    fTable_Si : ARRAY[0..755, 0..2] OF LREAL := [
        10.0000, -9999, 3.94851,
        10.1617, -9999, 3.95531,
        10.3261, -9999, 3.96212,
        10.4931, -9999, 3.96894,
        10.6628, -9999, 3.97577,
        10.8353, -9999, 3.98262,
        11.0105, -9999, 3.98948,
        11.1886, -9999, 3.99635,
        11.3696, -9999, 4.00322,
        11.5535, -9999, 4.01012,
        11.7404, -9999, 4.01702,
        11.9303, -9999, 4.02394,
        12.1232, -9999, 4.00019,
        12.3193, -9999, 3.95930,
        12.5186, -9999, 3.91883,
        12.7210, -9999, 3.87876,
        12.9268, -9999, 3.83911,
        13.1359, -9999, 3.79987,
        13.3483, -9999, 3.76102,
        13.5642, -9999, 3.72257,
        13.7836, -9999, 3.68452,
        14.0066, -9999, 3.64513,
        14.2331, -9999, 3.55020,
        14.4633, -9999, 3.45774,
        14.6972, -9999, 3.36769,
        14.9350, -9999, 3.27998,
        15.1765, -9999, 3.19455,
        15.4220, -9999, 3.11136,
        15.6714, -9999, 3.03032,
        15.9249, -9999, 2.95140,
        16.1825, -9999, 2.83114,
        16.4442, -9999, 2.69869,
        16.7102, -9999, 2.57244,
        16.9805, -9999, 2.45210,
        17.2551, -9999, 2.33738,
        17.5342, -9999, 2.22803,
        17.8178, -9999, 2.12380,
        18.1060, -9999, 1.97554,
        18.3988, -9999, 1.76138,
        18.6964, -9999, 1.57043,
        18.9988, -9999, 1.40019,
        19.3061, -9999, 1.24840,
        19.6184, -9999, 1.11306,
        19.9357, -9999, 0.992396,
        20.2581, -9999, 0.862336,
        20.5858, -9999, 0.753564,
        20.9187, -9999, 0.698871,
        21.2571, -9999, 0.648148,
        21.6009, -9999, 0.602543,
        21.9503, -9999, 0.561516,
        22.3053, -9999, 0.523281,
        22.6661, -9999, 0.496895,
        23.0327, -9999, 0.478071,
        23.4052, -9999, 0.459962,
        23.7838, -9999, 0.442538,
        24.1685, -9999, 0.425774,
        24.5594, -9999, 0.413096,
        24.9566, -9999, 0.403041,
        25.3602, -9999, 0.393231,
        25.7704, -9999, 0.383660,
        26.1872, -9999, 0.374321,
        26.6108, -9999, 0.365210,
        27.0412, -9999, 0.366288,
        27.4786, -9999, 0.367374,
        27.9230, -9999, 0.368463,
        28.3747, -9999, 0.369555,
        28.8336, -9999, 0.370650,
        29.3000, 3.83380, 0.371749,
        29.7739, 3.80691, 0.372851,
        30.2554, 3.78097, 0.373956,
        30.7448, 3.75582, 0.375064,
        31.2421, 3.73048, 0.376176,
        31.7474, 3.70550, 0.378088,
        32.2609, 3.68147, 0.381996,
        32.7827, 3.65905, 0.385945,
        33.3129, 3.63764, 0.389935,
        33.8517, 3.61703, 0.393965,
        34.3992, 3.59711, 0.398038,
        34.9556, 3.57779, 0.402152,
        35.5210, 3.55900, 0.406309,
        36.0955, 3.54071, 0.410509,
        36.6793, 3.52286, 0.414753,
        37.2726, 3.50545, 0.419040,
        37.8754, 3.48848, 0.423372,
        38.4880, 3.47200, 0.427748,
        39.1106, 3.45628, 0.432170,
        39.7431, 3.44176, 0.435537,
        40.3860, 3.42689, 0.437136,
        41.0392, 3.41050, 0.438741,
        41.7029, 3.39378, 0.440351,
        42.3774, 3.37667, 0.441968,
        43.0629, 3.35917, 0.443590,
        43.7594, 3.34130, 0.445218,
        44.4671, 3.32304, 0.446852,
        45.1864, 3.30440, 0.448493,
        45.9172, 3.28549, 0.450139,
        46.6599, 3.26615, 0.451198,
        47.4146, 3.24599, 0.451979,
        48.1815, 3.22476, 0.452762,
        48.9608, 3.20267, 0.453547,
        49.7527, 3.17964, 0.454332,
        50.5574, 3.15558, 0.455119,
        51.3751, 3.13042, 0.455908,
        52.2061, 3.10325, 0.456698,
        53.0505, 3.07444, 0.458301,
        53.9085, 3.04507, 0.461948,
        54.7804, 3.01545, 0.465624,
        55.6665, 2.98498, 0.469328,
        56.5668, 2.95338, 0.473062,
        57.4817, 2.92040, 0.476826,
        58.4115, 2.88519, 0.480620,
        59.3562, 2.84598, 0.484444,
        60.3163, 2.80606, 0.494947,
        61.2918, 2.76788, 0.506504,
        62.2832, 2.73042, 0.518332,
        63.2906, 2.69333, 0.530436,
        64.3142, 2.65696, 0.542822,
        65.3545, 2.62418, 0.554884,
        66.4115, 2.58874, 0.558968,
        67.4857, 2.54971, 0.563081,
        68.5772, 2.50917, 0.567224,
        69.6864, 2.46935, 0.571398,
        70.8135, 2.43129, 0.566814,
        71.9588, 2.38275, 0.552979,
        73.1227, 2.32504, 0.539483,
        74.3054, 2.26322, 0.526316,
        75.5072, 2.19828, 0.504782,
        76.7285, 2.11635, 0.477417,
        77.9695, 2.01618, 0.451535,
        79.2306, 1.90170, 0.427364,
        80.5121, 1.77437, 0.422623,
        81.8143, 1.64458, 0.417936,
        83.1376, 1.50518, 0.413300,
        84.4823, 1.34727, 0.409326,
        85.8487, 1.17621, 0.415946,
        87.2373, 0.995339, 0.422674,
        88.6483, 0.794497, 0.429510,
        90.0821, 0.568059, 0.436457,
        91.5391, 0.306962, 0.444926,
        93.0197, 0.00161588, 0.456528,
        94.5242, -0.366911, 0.468434,
        96.0530, -0.841388, 0.480650,
        97.6066, -1.52605, 0.495035,
        99.1853, -2.88115, 0.517644,
        99.5000, -3.50392, 0.522228,
        99.5240, -3.56793, 0.517644,
        99.5490, -3.65086, 0.517841,
        99.5760, -3.74861, 0.521284,
        99.6010, -3.84977, 0.535297,
        99.6260, -3.95788, 0.552022,
        99.6490, -4.07048, 0.581748,
        99.6760, -4.21370, 0.630001,
        99.6990, -4.33738, 0.708784,
        99.7260, -4.47439, 0.813415,
        99.7490, -4.57087, 0.941569,
        99.7750, -4.65499, 1.07721,
        99.8260, -4.76959, 1.37513,
        99.8510, -4.79109, 1.52203,
        99.8750, -4.78699, 1.65993,
        99.8990, -4.76674, 1.77995,
        99.9260, -4.73984, 1.87968,
        99.9510, -4.72571, 1.97448,
        99.9740, -4.69897, 2.05815,
        100.000, -4.67405, 2.13311,
        100.030, -4.65490, 2.20171,
        100.120, -4.60024, 2.41667,
        100.180, -4.60059, 2.49729,
        100.220, -4.62085, 2.58505,
        100.250, -4.64510, 2.62089,
        100.280, -4.70275, 2.67241,
        100.300, -4.73916, 2.73072,
        100.350, -4.82406, 2.91360,
        100.380, -4.87754, 3.01959,
        100.450, -4.89461, 3.39622,
        100.480, -4.89177, 3.52655,
        100.500, -4.87133, 3.64732,
        100.550, -4.80557, 3.86847,
        100.600, -4.71048, 4.10668,
        100.620, -4.63514, 4.23678,
        100.680, -4.54337, 4.36464,
        100.700, -4.48607, 4.49509,
        100.750, -4.33702, 4.75764,
        100.770, -4.23325, 4.85961,
        100.800, -4.07337, 4.94637,
        100.850, -3.81798, 5.07430,
        100.900, -3.56548, 5.12335,
        101.000, -3.15785, 5.13032,
        101.020, -3.08861, 5.12048,
        101.250, -2.52100, 5.15904,
        101.320, -2.30405, 5.19959,
        101.380, -2.08534, 5.20146,
        101.400, -2.00971, 5.18989,
        101.450, -1.81270, 5.13442,
        101.500, -1.65152, 5.02977,
        101.600, -1.41105, 4.78618,
        101.630, -1.36359, 4.72648,
        101.650, -1.35292, 4.65861,
        101.750, -1.25455, 4.44125,
        101.820, -1.21389, 4.30165,
        101.880, -1.19458, 4.18620,
        101.900, -1.20985, 4.13288,
        101.950, -1.20581, 4.08850,
        102.000, -1.19801, 3.97606,
        102.030, -1.22710, 3.93010,
        102.050, -1.24904, 3.89784,
        102.100, -1.28103, 3.86731,
        102.150, -1.30990, 3.80579,
        102.180, -1.33991, 3.78427,
        102.250, -1.39700, 3.76802,
        102.300, -1.42608, 3.74849,
        102.350, -1.46728, 3.74261,
        102.400, -1.50309, 3.76084,
        102.450, -1.52538, 3.79386,
        102.530, -1.50608, 3.87484,
        102.550, -1.48153, 3.89373,
        102.600, -1.42009, 3.90179,
        102.650, -1.36279, 3.88239,
        102.700, -1.31820, 3.83958,
        102.780, -1.29202, 3.76416,
        102.880, -1.29963, 3.67993,
        102.950, -1.32951, 3.64539,
        103.000, -1.34633, 3.63286,
        103.120, -1.36198, 3.65919,
        103.200, -1.32264, 3.65521,
        103.280, -1.27117, 3.62578,
        103.320, -1.25882, 3.57767,
        103.350, -1.24200, 3.56029,
        103.430, -1.23327, 3.47903,
        103.450, -1.26147, 3.44200,
        103.550, -1.32267, 3.37538,
        103.600, -1.36022, 3.35329,
        103.620, -1.37658, 3.35242,
        103.700, -1.42690, 3.33036,
        103.800, -1.48061, 3.33205,
        103.880, -1.50969, 3.33940,
        104.000, -1.53630, 3.33472,
        104.100, -1.56167, 3.31576,
        104.220, -1.62193, 3.27368,
        104.280, -1.65400, 3.27417,
        104.430, -1.72694, 3.28606,
        104.470, -1.75387, 3.27978,
        104.500, -1.76829, 3.28791,
        104.530, -1.78693, 3.28885,
        104.570, -1.80294, 3.29751,
        104.650, -1.83679, 3.30856,
        104.730, -1.87270, 3.30556,
        104.750, -1.88124, 3.31109,
        104.800, -1.90801, 3.30176,
        104.900, -1.98706, 3.33116,
        104.930, -2.00067, 3.33359,
        104.950, -2.00298, 3.34991,
        105.030, -2.04570, 3.36298,
        105.150, -2.11934, 3.39504,
        105.180, -2.13949, 3.40977,
        105.250, -2.17952, 3.43515,
        105.320, -2.21343, 3.47153,
        105.350, -2.23848, 3.47688,
        105.430, -2.28483, 3.52378,
        105.500, -2.32999, 3.56457,
        105.550, -2.35832, 3.60198,
        105.600, -2.38578, 3.64781,
        105.630, -2.39089, 3.66569,
        105.750, -2.44861, 3.77644,
        105.780, -2.45326, 3.79743,
        105.850, -2.48245, 3.88408,
        105.870, -2.48052, 3.91584,
        105.970, -2.42689, 4.01616,
        106.030, -2.39972, 4.04717,
        106.070, -2.38240, 4.06604,
        106.100, -2.37398, 4.06874,
        106.230, -2.38361, 4.11947,
        106.270, -2.37996, 4.15308,
        106.320, -2.37462, 4.16809,
        106.400, -2.36004, 4.21391,
        106.430, -2.36196, 4.22064,
        106.450, -2.36509, 4.23983,
        106.550, -2.33925, 4.28215,
        106.620, -2.33379, 4.30894,
        106.650, -2.33507, 4.32546,
        106.700, -2.32865, 4.34622,
        106.750, -2.32543, 4.37918,
        106.800, -2.31100, 4.39528,
        106.870, -2.30275, 4.43789,
        106.920, -2.28031, 4.45074,
        106.970, -2.27262, 4.47446,
        107.000, -2.25035, 4.47193,
        107.150, -2.24976, 4.52075,
        107.170, -2.23267, 4.52195,
        107.200, -2.22431, 4.53560,
        107.280, -2.22372, 4.53468,
        107.300, -2.22218, 4.54692,
        107.320, -2.21789, 4.54827,
        107.350, -2.21747, 4.55993,
        107.400, -2.22568, 4.56521,
        107.420, -2.21201, 4.58499,
        107.500, -2.21196, 4.60002,
        107.530, -2.21439, 4.60834,
        107.550, -2.21478, 4.62406,
        107.580, -2.20227, 4.63210,
        107.600, -2.20862, 4.62922,
        107.620, -2.19987, 4.64804,
        107.670, -2.19745, 4.66695,
        107.730, -2.18227, 4.67472,
        107.750, -2.19300, 4.68717,
        107.850, -2.17068, 4.70239,
        107.880, -2.18424, 4.71832,
        107.930, -2.18294, 4.73505,
        107.950, -2.19199, 4.75539,
        108.070, -2.15772, 4.79660,
        108.220, -2.13084, 4.82955,
        108.280, -2.11240, 4.85593,
        108.420, -2.08897, 4.88059,
        108.450, -2.08958, 4.88346,
        108.520, -2.07611, 4.91320,
        108.570, -2.06068, 4.91793,
        108.600, -2.05985, 4.93016,
        108.730, -2.02793, 4.92866,
        108.830, -2.03087, 4.94162,
        108.900, -2.01993, 4.96783,
        109.000, -1.99875, 4.97239,
        109.030, -1.99361, 4.97267,
        109.070, -1.99579, 4.95935,
        109.120, -2.00066, 4.97576,
        109.200, -2.00421, 4.98276,
        109.250, -1.99981, 4.99897,
        109.270, -1.98698, 4.98829,
        109.350, -2.00603, 4.99135,
        109.380, -2.00850, 4.98316,
        109.400, -2.01211, 4.99342,
        109.430, -2.02183, 4.98967,
        109.450, -2.01515, 5.00593,
        109.530, -2.04292, 5.01580,
        109.550, -2.03376, 5.03141,
        109.570, -2.03838, 5.02656,
        109.600, -2.03677, 5.04483,
        109.620, -2.03705, 5.03873,
        109.670, -2.02773, 5.05325,
        109.800, -2.05572, 5.08673,
        109.970, -2.05841, 5.12220,
        110.000, -2.08477, 5.13791,
        110.500, -2.08318, 5.28267,
        111.000, -2.07105, 5.45779,
        111.500, -2.02987, 5.61544,
        112.500, -1.94845, 5.85909,
        114.000, -1.92517, 6.16450,
        114.500, -1.96395, 6.33338,
        115.000, -1.98987, 6.51862,
        115.500, -1.96320, 6.72312,
        117.000, -1.77809, 7.40254,
        117.500, -1.61173, 7.59488,
        118.000, -1.45934, 7.77180,
        118.500, -1.28616, 7.87553,
        119.000, -1.13984, 8.02234,
        119.500, -0.959918, 8.05843,
        121.433, -0.578394, 8.42371,
        121.500, -0.573231, 8.43660,
        122.000, -0.405651, 8.51447,
        123.500, -0.0264126, 8.67192,
        124.000, 0.0779155, 8.69958,
        124.500, 0.171345, 8.77704,
        125.000, 0.293945, 8.78726,
        127.000, 0.572464, 9.00076,
        127.500, 0.671836, 9.04215,
        128.500, 0.827038, 9.19455,
        129.500, 0.995074, 9.33439,
        130.000, 1.11832, 9.43724,
        131.500, 1.53131, 9.68832,
        133.000, 2.07611, 9.80683,
        133.500, 2.28741, 9.78221,
        134.500, 2.61972, 9.60861,
        136.000, 2.84736, 9.24827,
        136.500, 2.87943, 9.17385,
        137.000, 2.87745, 9.11857,
        137.500, 2.85152, 9.03612,
        139.500, 2.83348, 9.09883,
        140.000, 2.84307, 9.12631,
        140.500, 2.88384, 9.18357,
        141.500, 3.00310, 9.19764,
        142.000, 3.03093, 9.17508,
        142.500, 3.03358, 9.18522,
        143.000, 3.03374, 9.17393,
        144.000, 3.03215, 9.32209,
        145.000, 3.09900, 9.41818,
        145.500, 3.16288, 9.49844,
        146.000, 3.22259, 9.51997,
        146.500, 3.28049, 9.57995,
        147.000, 3.34172, 9.60862,
        147.500, 3.41479, 9.66258,
        148.000, 3.48151, 9.67350,
        148.500, 3.56199, 9.71113,
        149.500, 3.68256, 9.71835,
        150.000, 3.70254, 9.69979,
        150.500, 3.68373, 9.74096,
        151.000, 3.69207, 9.84710,
        151.500, 3.76904, 10.0037,
        152.000, 3.94900, 10.1180,
        152.500, 4.15147, 10.1431,
        153.500, 4.47402, 9.96424,
        154.500, 4.52214, 9.69132,
        155.000, 4.47788, 9.64167,
        155.500, 4.41664, 9.63644,
        156.000, 4.38177, 9.66128,
        156.500, 4.35929, 9.73288,
        157.500, 4.39020, 9.79855,
        158.000, 4.36737, 9.87036,
        158.500, 4.42951, 9.99628,
        159.000, 4.48663, 9.99841,
        160.000, 4.57954, 10.1071,
        162.500, 4.84589, 10.5019,
        163.500, 5.05409, 10.6336,
        164.500, 5.27583, 10.7324,
        165.500, 5.50795, 10.7656,
        166.500, 5.73389, 10.8239,
        167.000, 5.79695, 10.7800,
        167.500, 5.86489, 10.9015,
        169.000, 6.35522, 10.9520,
        170.000, 6.66644, 10.9210,
        171.500, 7.13398, 10.7554,
        172.000, 7.24279, 10.5495,
        172.500, 7.29281, 10.5369,
        173.000, 7.38343, 10.4391,
        173.500, 7.52303, 10.4208,
        174.000, 7.60600, 10.1923,
        174.500, 7.64212, 10.1249,
        175.000, 7.66842, 9.98038,
        176.000, 7.68591, 9.82584,
        176.500, 7.67332, 9.72546,
        177.000, 7.68563, 9.66145,
        178.000, 7.67511, 9.60542,
        178.500, 7.69740, 9.51565,
        179.000, 7.64095, 9.49283,
        179.500, 7.63925, 9.43704,
        179.990, 7.55398, 9.49765,
        182.901, 7.85149, 9.42072,
        185.859, 7.94847, 9.34442,
        188.866, 8.10574, 9.26640,
        191.920, 8.27005, 9.17918,
        195.025, 8.43202, 9.09278,
        198.179, 8.59128, 9.00719,
        201.384, 8.74251, 8.92241,
        204.641, 8.88646, 8.85010,
        207.951, 9.03960, 8.78533,
        211.315, 9.19861, 8.72104,
        214.733, 9.36085, 8.65722,
        218.206, 9.53668, 8.59386,
        221.735, 9.72509, 8.52313,
        225.322, 9.90451, 8.41115,
        228.966, 10.0644, 8.30065,
        232.669, 10.2142, 8.19159,
        236.432, 10.3574, 8.08397,
        240.257, 10.4958, 7.97776,
        244.143, 10.6314, 7.87295,
        248.091, 10.7716, 7.76952,
        252.104, 10.9063, 7.65024,
        256.182, 11.0283, 7.53005,
        260.325, 11.1426, 7.41174,
        264.536, 11.2509, 7.29529,
        268.814, 11.3543, 7.18067,
        273.162, 11.4535, 7.06784,
        277.580, 11.5489, 6.95680,
        282.070, 11.6411, 6.84750,
        286.632, 11.7306, 6.73991,
        291.268, 11.8181, 6.63402,
        295.979, 11.9057, 6.52979,
        300.767, 11.9918, 6.42157,
        305.631, 12.0733, 6.31071,
        310.575, 12.1486, 6.20175,
        315.598, 12.2203, 6.09469,
        320.702, 12.2889, 5.98947,
        325.890, 12.3551, 5.88607,
        331.161, 12.4191, 5.78445,
        336.517, 12.4812, 5.68459,
        341.960, 12.5420, 5.58645,
        347.491, 12.6018, 5.49000,
        353.111, 12.6614, 5.39523,
        358.822, 12.7222, 5.30208,
        364.626, 12.7889, 5.21055,
        370.523, 12.8576, 5.10056,
        376.516, 12.9142, 4.98768,
        382.606, 12.9608, 4.87731,
        388.795, 13.0027, 4.76937,
        395.083, 13.0407, 4.66382,
        401.473, 13.0753, 4.56061,
        407.967, 13.1069, 4.45967,
        414.565, 13.1360, 4.36098,
        421.270, 13.1628, 4.26447,
        428.084, 13.1876, 4.17009,
        435.008, 13.2107, 4.07781,
        442.044, 13.2322, 3.98756,
        449.194, 13.2527, 3.89931,
        456.459, 13.2727, 3.81302,
        463.842, 13.2933, 3.72727,
        471.344, 13.3117, 3.63809,
        478.968, 13.3260, 3.55105,
        486.715, 13.3375, 3.46608,
        494.587, 13.3472, 3.38316,
        502.587, 13.3552, 3.30221,
        510.715, 13.3617, 3.22320,
        518.976, 13.3670, 3.14609,
        527.370, 13.3711, 3.07081,
        535.900, 13.3742, 2.99734,
        544.567, 13.3764, 2.92563,
        553.375, 13.3779, 2.85563,
        562.326, 13.3789, 2.78730,
        571.421, 13.3797, 2.72061,
        580.663, 13.3815, 2.65552,
        590.055, 13.3832, 2.58813,
        599.599, 13.3823, 2.52006,
        609.297, 13.3786, 2.45378,
        619.151, 13.3731, 2.38925,
        629.166, 13.3663, 2.32641,
        639.342, 13.3582, 2.26522,
        649.683, 13.3491, 2.20565,
        660.191, 13.3390, 2.14764,
        670.869, 13.3278, 2.09115,
        681.720, 13.3158, 2.03616,
        692.746, 13.3006, 1.98261,
        703.951, 13.2845, 1.93392,
        715.336, 13.2706, 1.88812,
        726.906, 13.2578, 1.84339,
        738.664, 13.2453, 1.79973,
        750.611, 13.2332, 1.75710,
        762.751, 13.2215, 1.71548,
        775.088, 13.2102, 1.67484,
        787.625, 13.1996, 1.63517,
        800.364, 13.1912, 1.59508,
        813.309, 13.1807, 1.55256,
        826.464, 13.1685, 1.51118,
        839.831, 13.1555, 1.47089,
        853.415, 13.1418, 1.43168,
        867.218, 13.1278, 1.39352,
        881.245, 13.1136, 1.35637,
        895.498, 13.1001, 1.32021,
        909.982, 13.0874, 1.28196,
        924.700, 13.0717, 1.24308,
        939.656, 13.0542, 1.20538,
        954.855, 13.0353, 1.16882,
        970.299, 13.0154, 1.13337,
        985.992, 12.9946, 1.09899,
        1001.94, 12.9729, 1.06561,
        1018.15, 12.9502, 1.03318,
        1034.61, 12.9266, 1.00174,
        1051.35, 12.9020, 0.971249,
        1068.35, 12.8761, 0.941688,
        1085.63, 12.8487, 0.913028,
        1103.19, 12.8192, 0.887547,
        1121.03, 12.7911, 0.864407,
        1139.17, 12.7632, 0.841817,
        1157.59, 12.7350, 0.819826,
        1176.31, 12.7063, 0.798411,
        1195.34, 12.6771, 0.777531,
        1214.67, 12.6470, 0.757139,
        1234.32, 12.6159, 0.737234,
        1254.28, 12.5837, 0.717856,
        1274.57, 12.5503, 0.698989,
        1295.19, 12.5156, 0.680609,
        1316.13, 12.4792, 0.662552,
        1337.42, 12.4409, 0.644954,
        1359.05, 12.4006, 0.627806,
        1381.04, 12.3579, 0.611117,
        1403.37, 12.3125, 0.594814,
        1426.07, 12.2640, 0.578892,
        1449.14, 12.2120, 0.563357,
        1472.58, 12.1559, 0.548240,
        1496.39, 12.0950, 0.533519,
        1520.60, 12.0284, 0.518512,
        1545.19, 11.9546, 0.503884,
        1570.18, 11.8721, 0.489627,
        1595.58, 11.7790, 0.475781,
        1621.39, 11.6727, 0.462322,
        1647.61, 11.5493, 0.449240,
        1674.26, 11.4029, 0.436529,
        1701.34, 11.2243, 0.424180,
        1728.86, 10.9982, 0.412181,
        1756.82, 10.6935, 0.399995,
        1785.24, 10.2377, 0.388066,
        1814.11, 9.37942, 0.376400,
        1815, 9.33435, 0.376049,
        1838.80, 2.82013, 0.366843,
        1839, 2.82204, 2.26608,
        1838.90, 7.96957, 4.15773,
        1860, 9.34866, 4.09222,
        1890.08, 10.4859, 4.00184,
        1920.65, 11.1017, 3.91340,
        1951.72, 11.5305, 3.82687,
        1983.29, 11.8609, 3.74224,
        2015.37, 12.1301, 3.65896,
        2047.96, 12.3571, 3.57698,
        2081.09, 12.5533, 3.49664,
        2114.75, 12.7254, 3.41523,
        2148.95, 12.8775, 3.33521,
        2183.71, 13.0131, 3.25641,
        2219.03, 13.1350, 3.17868,
        2254.92, 13.2452, 3.10245,
        2291.39, 13.3453, 3.02741,
        2328.45, 13.4369, 2.95359,
        2366.11, 13.5205, 2.88121,
        2404.38, 13.5972, 2.80993,
        2443.27, 13.6676, 2.74011,
        2482.79, 13.7324, 2.67152,
        2522.95, 13.7921, 2.60424,
        2563.75, 13.8472, 2.53844,
        2605.22, 13.8981, 2.47374,
        2647.36, 13.9449, 2.41045,
        2690.18, 13.9882, 2.34854,
        2733.69, 14.0282, 2.28769,
        2777.90, 14.0651, 2.22827,
        2822.83, 14.0991, 2.17014,
        2868.49, 14.1305, 2.11320,
        2914.89, 14.1594, 2.05756,
        2962.03, 14.1859, 2.00307,
        3009.94, 14.2104, 1.94988,
        3058.62, 14.2329, 1.89788,
        3108.09, 14.2535, 1.84703,
        3158.37, 14.2723, 1.79742,
        3209.45, 14.2894, 1.74890,
        3261.36, 14.3051, 1.70154,
        3314.11, 14.3194, 1.65534,
        3367.71, 14.3322, 1.61015,
        3422.18, 14.3438, 1.56612,
        3477.53, 14.3542, 1.52314,
        3533.78, 14.3635, 1.48119,
        3590.94, 14.3718, 1.44032,
        3649.02, 14.3791, 1.40039,
        3708.04, 14.3855, 1.36149,
        3768.01, 14.3910, 1.32359,
        3828.96, 14.3957, 1.28658,
        3890.89, 14.3997, 1.25056,
        3953.82, 14.4029, 1.21543,
        4017.77, 14.4055, 1.18120,
        4082.75, 14.4075, 1.14788,
        4148.79, 14.4089, 1.11537,
        4215.89, 14.4097, 1.08375,
        4284.08, 14.4101, 1.05295,
        4353.37, 14.4100, 1.02294,
        4423.78, 14.4094, 0.993744,
        4495.33, 14.4085, 0.965295,
        4568.04, 14.4071, 0.937606,
        4641.93, 14.4054, 0.910663,
        4717.01, 14.4034, 0.884415,
        4793.30, 14.4011, 0.858896,
        4870.83, 14.3984, 0.834074,
        4949.61, 14.3956, 0.809917,
        5029.67, 14.3925, 0.786429,
        5111.02, 14.3891, 0.763535,
        5193.68, 14.3856, 0.741289,
        5277.69, 14.3818, 0.719672,
        5363.05, 14.3779, 0.698635,
        5449.79, 14.3739, 0.678189,
        5537.94, 14.3697, 0.658294,
        5627.51, 14.3654, 0.638950,
        5718.53, 14.3609, 0.620147,
        5811.02, 14.3564, 0.601873,
        5905.01, 14.3517, 0.584116,
        6000.52, 14.3470, 0.566843,
        6097.57, 14.3422, 0.550055,
        6196.20, 14.3374, 0.533751,
        6296.42, 14.3325, 0.517913,
        6349, 14.3300, 0.509889,
        6432, 14.3259, 0.497536,
        6536.03, 14.3209, 0.482727,
        6641.75, 14.3159, 0.468336,
        6749.17, 14.3109, 0.454339,
        6858.33, 14.3059, 0.440746,
        6969.26, 14.3008, 0.427550,
        7081.98, 14.2958, 0.414725,
        7196.53, 14.2907, 0.402271,
        7312.93, 14.2857, 0.390179,
        7431.21, 14.2806, 0.378427,
        7551.40, 14.2756, 0.367020,
        7673.54, 14.2706, 0.355946,
        7797.65, 14.2657, 0.345189,
        7923.77, 14.2607, 0.334747,
        8051.94, 14.2558, 0.324605,
        8182.17, 14.2510, 0.314762,
        8314.51, 14.2461, 0.305207,
        8448.99, 14.2414, 0.295929,
        8585.64, 14.2366, 0.286926,
        8724.51, 14.2319, 0.278183,
        8865.62, 14.2273, 0.269697,
        9009.02, 14.2227, 0.261465,
        9154.73, 14.2181, 0.253469,
        9302.80, 14.2136, 0.245713,
        9453.27, 14.2091, 0.238188,
        9606.17, 14.2047, 0.230880,
        9761.54, 14.2004, 0.223790,
        9919.42, 14.1961, 0.216911,
        10079.9, 14.1919, 0.210235,
        10242.9, 14.1877, 0.203758,
        10408.6, 14.1836, 0.197474,
        10576.9, 14.1795, 0.191376,
        10748.0, 14.1756, 0.185461,
        10921.8, 14.1716, 0.179721,
        11098.5, 14.1677, 0.174154,
        11278.0, 14.1639, 0.168752,
        11460.4, 14.1602, 0.163513,
        11645.8, 14.1565, 0.158430,
        11834.1, 14.1528, 0.153500,
        12025.5, 14.1492, 0.148717,
        12220.0, 14.1457, 0.144079,
        12417.7, 14.1423, 0.139580,
        12618.5, 14.1389, 0.135216,
        12822.6, 14.1355, 0.130984,
        13030.0, 14.1322, 0.126879,
        13240.8, 14.1290, 0.122899,
        13454.9, 14.1258, 0.119038,
        13672.6, 14.1227, 0.115294,
        13893.7, 14.1197, 0.111664,
        14118.4, 14.1167, 0.108143,
        14346.8, 14.1137, 0.104730,
        14578.8, 14.1108, 0.101419,
        14814.6, 14.1080, 0.0982093,
        15054.2, 14.1052, 0.0950968,
        15297.7, 14.1025, 0.0920790,
        15545.2, 14.0998, 0.0891530,
        15796.6, 14.0972, 0.0863160,
        16052.1, 14.0946, 0.0835654,
        16311.7, 14.0921, 0.0808987,
        16575.5, 14.0896, 0.0783132,
        16843.6, 14.0872, 0.0758067,
        17116.1, 14.0848, 0.0733767,
        17392.9, 14.0825, 0.0710210,
        17674.2, 14.0802, 0.0687373,
        17960.1, 14.0780, 0.0665234,
        18250.6, 14.0758, 0.0643773,
        18545.8, 14.0736, 0.0622970,
        18845.7, 14.0715, 0.0602804,
        19150.5, 14.0695, 0.0583256,
        19460.3, 14.0675, 0.0564308,
        19775.0, 14.0655, 0.0545942,
        20094.9, 14.0636, 0.0528124,
        20419.9, 14.0617, 0.0510884,
        20750.2, 14.0598, 0.0494193,
        21085.8, 14.0580, 0.0478034,
        21426.8, 14.0562, 0.0462390,
        21773.4, 14.0545, 0.0447245,
        22125.6, 14.0528, 0.0432583,
        22483.4, 14.0511, 0.0418390,
        22847.1, 14.0495, 0.0404650,
        23216.6, 14.0479, 0.0391349,
        23592.1, 14.0463, 0.0378475,
        23973.7, 14.0448, 0.0366013,
        24361.5, 14.0433, 0.0353950,
        24755.5, 14.0419, 0.0342274,
        25155.9, 14.0405, 0.0330973,
        25562.8, 14.0391, 0.0320035,
        25976.2, 14.0377, 0.0309448,
        26396.4, 14.0364, 0.0299202,
        26823.3, 14.0351, 0.0289286,
        27257.2, 14.0338, 0.0279690,
        27698.0, 14.0326, 0.0270403,
        28146.0, 14.0314, 0.0261415,
        28601.3, 14.0302, 0.0252718,
        29063.9, 14.0291, 0.0244301,
        29533.9, 14.0279, 0.0236157,
        30000.0, 14.0269, 0.0228464
    ];

END_VAR


(* WARNING: This file is auto-generated. Do not modify it.*)
(* Get correct table *)


IF sTableName = 'Ge' THEN
    iRowSize := ADR(fTable_Ge[1,0]) - ADR(fTable_Ge[0,0]);
    iRowCount := 505;
    fRow1 := ADR(fTable_Ge[0, 0]);
    fTableLookupLow := 10.0000;
    fTableLookupHigh := 30000.0;
ELSIF sTableName = 'C' THEN
    iRowSize := ADR(fTable_C[1,0]) - ADR(fTable_C[0,0]);
    iRowCount := 501;
    fRow1 := ADR(fTable_C[0, 0]);
    fTableLookupLow := 10.0000;
    fTableLookupHigh := 30000.0;
ELSIF sTableName = 'Al' THEN
    iRowSize := ADR(fTable_Al[1,0]) - ADR(fTable_Al[0,0]);
    iRowCount := 503;
    fRow1 := ADR(fTable_Al[0, 0]);
    fTableLookupLow := 10.0000;
    fTableLookupHigh := 30000.0;
ELSIF sTableName = 'Be' THEN
    iRowSize := ADR(fTable_Be[1,0]) - ADR(fTable_Be[0,0]);
    iRowCount := 723;
    fRow1 := ADR(fTable_Be[0, 0]);
    fTableLookupLow := 10.0000;
    fTableLookupHigh := 30000.0;
ELSIF sTableName = 'Si' THEN
    iRowSize := ADR(fTable_Si[1,0]) - ADR(fTable_Si[0,0]);
    iRowCount := 755;
    fRow1 := ADR(fTable_Si[0, 0]);
    fTableLookupLow := 10.0000;
    fTableLookupHigh := 30000.0;
ELSE
    bFound := FALSE;
    bError := TRUE;
    RETURN;
END_IF

bError := FALSE;
bFound := FALSE;

IF fEnergyEV < fTableLookupLow THEN
    RETURN;
ELSIF fEnergyEV > fTableLookupHigh THEN
    RETURN;
END_IF

FOR iRowIdx := 0 TO iRowCount - 1
DO
    fRow2 := fRow1 + iRowSize;
    IF fEnergyEV >= fRow1^[0] AND fEnergyEV <= fRow2^[0] THEN
        fEnergyEV_RowDelta := fRow2^[0] - fRow1^[0];
        IF fEnergyEV_RowDelta <= 0.0 THEN
            bFound := TRUE;
            bError := TRUE;
        ELSE

            // Interpolate output: f1
            fSlope := (fRow2^[1] - fRow1^[1]) / fEnergyEV_RowDelta;
            f1 := fRow1^[1] + fSlope * (fEnergyEV - fRow1^[0]);

            // Interpolate output: f2
            fSlope := (fRow2^[2] - fRow1^[2]) / fEnergyEV_RowDelta;
            f2 := fRow1^[2] + fSlope * (fEnergyEV - fRow1^[0]);
 
            bFound := TRUE;
            bError := FALSE;
        END_IF
        RETURN;
    END_IF
    fRow1 := fRow2;
END_FOR

END_FUNCTION_BLOCK

(* stored: Version 1.1.0.1, ProductVersion 3.1.4024.4
   POU FB_AbsorptionLUT: Id {bcc5442f-16ea-00be-b111-68f89e3450e2}, SpecialFunc None *)
